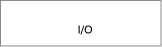
VISUALIZATION VISU_AxesIO  // 162x47
VAR_IN_OUT
	ref : AxesIO;
    widget : AxesIOWidget;
END_VAR
    Label (10,15 150x30), "I/O"
END_VISUALIZATION

(* stored: Version 1.1.0.1, ProductVersion 3.1.4018.5
   Visu VISU_AxesIO: Id {3c336157-4787-46e8-98d8-0a79d2f8a1cf} *)
